	                            // ==============================================================================
	                            // Segment [9]
	                            // ==============================================================================
	                            #tempCalAcc[9] := #tempJerk[9 - 1] * #tempX[9 - 1] + #tempCalAcc[9 - 1];
	                            #tempCalVel[9] := #tempJerk[9 - 1] * #tempX[9 - 1] * #tempX[9 - 1] / 2.0 + #tempCalAcc[9 - 1] * #tempX[9 - 1] + #tempCalVel[9 - 1];
	                            #tempCalPos[9] := #tempJerk[9 - 1] * #tempX[9 - 1] * #tempX[9 - 1] * #tempX[9 - 1] / 6.0 + #tempCalAcc[9 - 1] * #tempX[9 - 1] * #tempX[9 - 1] / 2.0 + #tempCalVel[9 - 1] * #tempX[9 - 1] + #tempCalPos[9 - 1];
	                            IF ABS_LREAL(#tempCalVel[9]) < 0.000000001 THEN
	                                #tempCalVel[9] := 0.0;
	                            END_IF;
	                            IF ABS_LREAL(#tempCalPos[9]) < 0.000000001 THEN
	                                #tempCalPos[9] := 0.0;
	                            END_IF;
	                            #tempA3[9] := #tempJerk[9] / 6.0;
	                            #tempA2[9] := #tempCalAcc[9] / 2.0;
	                            #tempA1[9] := #tempCalVel[9];
	                            #tempA0[9] := #tempCalPos[9];
	                            #tempCam^.Segment[9].a0 := #tempA0[9];
	                            #tempCam^.Segment[9].a1 := #tempA1[9];
	                            #tempCam^.Segment[9].a2 := #tempA2[9];
	                            #tempCam^.Segment[9].a3 := #tempA3[9];
	                            #tempCam^.Segment[9].a4 := 0.0;
	                            #tempCam^.Segment[9].a5 := 0.0;
	                            #tempCam^.Segment[9].a6 := 0.0;
	                            #tempCam^.Segment[9].xmax := #tempCam^.Segment[9 - 1].xmax + #tempX[9];
	                            #tempCam^.Segment[9].xmin := #tempCam^.Segment[9 - 1].xmax;
	                            #tempCam^.Segment[9].sineAmplitude := 0.0;
	                            #tempCam^.Segment[9].sinePeriod := 0.0;
	                            #tempCam^.Segment[9].sinePhase := 0.0;
	                            IF #tempX[9] = 0.0 THEN
	                                #tempCam^.ValidSegment[9] := FALSE;
	                            ELSE
	                                #tempCam^.ValidSegment[9] := TRUE;
	                            END_IF;

	                            // ==============================================================================
	                            // Segment [10]
	                            // ==============================================================================
	                            #tempCalAcc[10] := #tempJerk[10 - 1] * #tempX[10 - 1] + #tempCalAcc[10 - 1];
	                            #tempCalVel[10] := #tempJerk[10 - 1] * #tempX[10 - 1] * #tempX[10 - 1] / 2.0 + #tempCalAcc[10 - 1] * #tempX[10 - 1] + #tempCalVel[10 - 1];
	                            #tempCalPos[10] := #tempJerk[10 - 1] * #tempX[10 - 1] * #tempX[10 - 1] * #tempX[10 - 1] / 6.0 + #tempCalAcc[10 - 1] * #tempX[10 - 1] * #tempX[10 - 1] / 2.0 + #tempCalVel[10 - 1] * #tempX[10 - 1] + #tempCalPos[10 - 1];
	                            IF ABS_LREAL(#tempCalVel[10]) < 0.000000001 THEN
	                                #tempCalVel[10] := 0.0;
	                            END_IF;
	                            IF ABS_LREAL(#tempCalPos[10]) < 0.000000001 THEN
	                                #tempCalPos[10] := 0.0;
	                            END_IF;
	                            #tempA3[10] := #tempJerk[10] / 6.0;
	                            #tempA2[10] := #tempCalAcc[10] / 2.0;
	                            #tempA1[10] := #tempCalVel[10];
	                            #tempA0[10] := #tempCalPos[10];
	                            #tempCam^.Segment[10].a0 := #tempA0[10];
	                            #tempCam^.Segment[10].a1 := #tempA1[10];
	                            #tempCam^.Segment[10].a2 := #tempA2[10];
	                            #tempCam^.Segment[10].a3 := #tempA3[10];
	                            #tempCam^.Segment[10].a4 := 0.0;
	                            #tempCam^.Segment[10].a5 := 0.0;
	                            #tempCam^.Segment[10].a6 := 0.0;
	                            #tempCam^.Segment[10].xmax := #tempCam^.Segment[10 - 1].xmax + #tempX[10];
	                            #tempCam^.Segment[10].xmin := #tempCam^.Segment[10 - 1].xmax;
	                            #tempCam^.Segment[10].sineAmplitude := 0.0;
	                            #tempCam^.Segment[10].sinePeriod := 0.0;
	                            #tempCam^.Segment[10].sinePhase := 0.0;
	                            IF #tempX[10] = 0.0 THEN
	                                #tempCam^.ValidSegment[10] := FALSE;
	                            ELSE
	                                #tempCam^.ValidSegment[10] := TRUE;
	                            END_IF;

	                            // ==============================================================================
	                            // Segment [11]
	                            // ==============================================================================
	                            #tempCalAcc[11] := #tempJerk[11 - 1] * #tempX[11 - 1] + #tempCalAcc[11 - 1];
	                            #tempCalVel[11] := #tempJerk[11 - 1] * #tempX[11 - 1] * #tempX[11 - 1] / 2.0 + #tempCalAcc[11 - 1] * #tempX[11 - 1] + #tempCalVel[11 - 1];
	                            #tempCalPos[11] := #tempJerk[11 - 1] * #tempX[11 - 1] * #tempX[11 - 1] * #tempX[11 - 1] / 6.0 + #tempCalAcc[11 - 1] * #tempX[11 - 1] * #tempX[11 - 1] / 2.0 + #tempCalVel[11 - 1] * #tempX[11 - 1] + #tempCalPos[11 - 1];
	                            IF ABS_LREAL(#tempCalVel[11]) < 0.000000001 THEN
	                                #tempCalVel[11] := 0.0;
	                            END_IF;
	                            IF ABS_LREAL(#tempCalPos[11]) < 0.000000001 THEN
	                                #tempCalPos[11] := 0.0;
	                            END_IF;
	                            #tempA3[11] := #tempJerk[11] / 6.0;
	                            #tempA2[11] := #tempCalAcc[11] / 2.0;
	                            #tempA1[11] := #tempCalVel[11];
	                            #tempA0[11] := #tempCalPos[11];
	                            #tempCam^.Segment[11].a0 := #tempA0[11];
	                            #tempCam^.Segment[11].a1 := #tempA1[11];
	                            #tempCam^.Segment[11].a2 := #tempA2[11];
	                            #tempCam^.Segment[11].a3 := #tempA3[11];
	                            #tempCam^.Segment[11].a4 := 0.0;
	                            #tempCam^.Segment[11].a5 := 0.0;
	                            #tempCam^.Segment[11].a6 := 0.0;
	                            #tempCam^.Segment[11].xmax := #tempCam^.Segment[11 - 1].xmax + #tempX[11];
	                            #tempCam^.Segment[11].xmin := #tempCam^.Segment[11 - 1].xmax;
	                            #tempCam^.Segment[11].sineAmplitude := 0.0;
	                            #tempCam^.Segment[11].sinePeriod := 0.0;
	                            #tempCam^.Segment[11].sinePhase := 0.0;
	                            IF #tempX[11] = 0.0 THEN
	                                #tempCam^.ValidSegment[11] := FALSE;
	                            ELSE
	                                #tempCam^.ValidSegment[11] := TRUE;
	                            END_IF;

	                            // ==============================================================================
	                            // Segment [12]
	                            // ==============================================================================
	                            #tempCalAcc[12] := #tempJerk[12 - 1] * #tempX[12 - 1] + #tempCalAcc[12 - 1];
	                            #tempCalVel[12] := #tempJerk[12 - 1] * #tempX[12 - 1] * #tempX[12 - 1] / 2.0 + #tempCalAcc[12 - 1] * #tempX[12 - 1] + #tempCalVel[12 - 1];
	                            #tempCalPos[12] := #tempJerk[12 - 1] * #tempX[12 - 1] * #tempX[12 - 1] * #tempX[12 - 1] / 6.0 + #tempCalAcc[12 - 1] * #tempX[12 - 1] * #tempX[12 - 1] / 2.0 + #tempCalVel[12 - 1] * #tempX[12 - 1] + #tempCalPos[12 - 1];
	                            IF ABS_LREAL(#tempCalVel[12]) < 0.000000001 THEN
	                                #tempCalVel[12] := 0.0;
	                            END_IF;
	                            IF ABS_LREAL(#tempCalPos[12]) < 0.000000001 THEN
	                                #tempCalPos[12] := 0.0;
	                            END_IF;
	                            #tempA3[12] := #tempJerk[12] / 6.0;
	                            #tempA2[12] := #tempCalAcc[12] / 2.0;
	                            #tempA1[12] := #tempCalVel[12];
	                            #tempA0[12] := #tempCalPos[12];
	                            #tempCam^.Segment[12].a0 := #tempA0[12];
	                            #tempCam^.Segment[12].a1 := #tempA1[12];
	                            #tempCam^.Segment[12].a2 := #tempA2[12];
	                            #tempCam^.Segment[12].a3 := #tempA3[12];
	                            #tempCam^.Segment[12].a4 := 0.0;
	                            #tempCam^.Segment[12].a5 := 0.0;
	                            #tempCam^.Segment[12].a6 := 0.0;
	                            #tempCam^.Segment[12].xmax := #tempCam^.Segment[12 - 1].xmax + #tempX[12];
	                            #tempCam^.Segment[12].xmin := #tempCam^.Segment[12 - 1].xmax;
	                            #tempCam^.Segment[12].sineAmplitude := 0.0;
	                            #tempCam^.Segment[12].sinePeriod := 0.0;
	                            #tempCam^.Segment[12].sinePhase := 0.0;
	                            IF #tempX[12] = 0.0 THEN
	                                #tempCam^.ValidSegment[12] := FALSE;
	                            ELSE
	                                #tempCam^.ValidSegment[12] := TRUE;
	                            END_IF;

	                            // ==============================================================================
	                            // Segment [13]
	                            // ==============================================================================
	                            #tempCalAcc[13] := #tempJerk[13 - 1] * #tempX[13 - 1] + #tempCalAcc[13 - 1];
	                            #tempCalVel[13] := #tempJerk[13 - 1] * #tempX[13 - 1] * #tempX[13 - 1] / 2.0 + #tempCalAcc[13 - 1] * #tempX[13 - 1] + #tempCalVel[13 - 1];
	                            #tempCalPos[13] := #tempJerk[13 - 1] * #tempX[13 - 1] * #tempX[13 - 1] * #tempX[13 - 1] / 6.0 + #tempCalAcc[13 - 1] * #tempX[13 - 1] * #tempX[13 - 1] / 2.0 + #tempCalVel[13 - 1] * #tempX[13 - 1] + #tempCalPos[13 - 1];
	                            IF ABS_LREAL(#tempCalVel[13]) < 0.000000001 THEN
	                                #tempCalVel[13] := 0.0;
	                            END_IF;
	                            IF ABS_LREAL(#tempCalPos[13]) < 0.000000001 THEN
	                                #tempCalPos[13] := 0.0;
	                            END_IF;
	                            #tempA3[13] := #tempJerk[13] / 6.0;
	                            #tempA2[13] := #tempCalAcc[13] / 2.0;
	                            #tempA1[13] := #tempCalVel[13];
	                            #tempA0[13] := #tempCalPos[13];
	                            #tempCam^.Segment[13].a0 := #tempA0[13];
	                            #tempCam^.Segment[13].a1 := #tempA1[13];
	                            #tempCam^.Segment[13].a2 := #tempA2[13];
	                            #tempCam^.Segment[13].a3 := #tempA3[13];
	                            #tempCam^.Segment[13].a4 := 0.0;
	                            #tempCam^.Segment[13].a5 := 0.0;
	                            #tempCam^.Segment[13].a6 := 0.0;
	                            #tempCam^.Segment[13].xmax := #tempCam^.Segment[13 - 1].xmax + #tempX[13];
	                            #tempCam^.Segment[13].xmin := #tempCam^.Segment[13 - 1].xmax;
	                            #tempCam^.Segment[13].sineAmplitude := 0.0;
	                            #tempCam^.Segment[13].sinePeriod := 0.0;
	                            #tempCam^.Segment[13].sinePhase := 0.0;
	                            IF #tempX[13] = 0.0 THEN
	                                #tempCam^.ValidSegment[13] := FALSE;
	                            ELSE
	                                #tempCam^.ValidSegment[13] := TRUE;
	                            END_IF;

	                            // ==============================================================================
	                            // Segment [14]
	                            // ==============================================================================
	                            #tempCalAcc[14] := #tempJerk[14 - 1] * #tempX[14 - 1] + #tempCalAcc[14 - 1];
	                            #tempCalVel[14] := #tempJerk[14 - 1] * #tempX[14 - 1] * #tempX[14 - 1] / 2.0 + #tempCalAcc[14 - 1] * #tempX[14 - 1] + #tempCalVel[14 - 1];
	                            #tempCalPos[14] := #tempJerk[14 - 1] * #tempX[14 - 1] * #tempX[14 - 1] * #tempX[14 - 1] / 6.0 + #tempCalAcc[14 - 1] * #tempX[14 - 1] * #tempX[14 - 1] / 2.0 + #tempCalVel[14 - 1] * #tempX[14 - 1] + #tempCalPos[14 - 1];
	                            IF ABS_LREAL(#tempCalVel[14]) < 0.000000001 THEN
	                                #tempCalVel[14] := 0.0;
	                            END_IF;
	                            IF ABS_LREAL(#tempCalPos[14]) < 0.000000001 THEN
	                                #tempCalPos[14] := 0.0;
	                            END_IF;
	                            #tempA3[14] := #tempJerk[14] / 6.0;
	                            #tempA2[14] := #tempCalAcc[14] / 2.0;
	                            #tempA1[14] := #tempCalVel[14];
	                            #tempA0[14] := #tempCalPos[14];
	                            #tempCam^.Segment[14].a0 := #tempA0[14];
	                            #tempCam^.Segment[14].a1 := #tempA1[14];
	                            #tempCam^.Segment[14].a2 := #tempA2[14];
	                            #tempCam^.Segment[14].a3 := #tempA3[14];
	                            #tempCam^.Segment[14].a4 := 0.0;
	                            #tempCam^.Segment[14].a5 := 0.0;
	                            #tempCam^.Segment[14].a6 := 0.0;
	                            #tempCam^.Segment[14].xmax := #tempCam^.Segment[14 - 1].xmax + #tempX[14];
	                            #tempCam^.Segment[14].xmin := #tempCam^.Segment[14 - 1].xmax;
	                            #tempCam^.Segment[14].sineAmplitude := 0.0;
	                            #tempCam^.Segment[14].sinePeriod := 0.0;
	                            #tempCam^.Segment[14].sinePhase := 0.0;
	                            IF #tempX[14] = 0.0 THEN
	                                #tempCam^.ValidSegment[14] := FALSE;
	                            ELSE
	                                #tempCam^.ValidSegment[14] := TRUE;
	                            END_IF;

	                            // ==============================================================================
	                            // Segment [15]
	                            // ==============================================================================
	                            #tempCalAcc[15] := #tempJerk[15 - 1] * #tempX[15 - 1] + #tempCalAcc[15 - 1];
	                            #tempCalVel[15] := #tempJerk[15 - 1] * #tempX[15 - 1] * #tempX[15 - 1] / 2.0 + #tempCalAcc[15 - 1] * #tempX[15 - 1] + #tempCalVel[15 - 1];
	                            #tempCalPos[15] := #tempJerk[15 - 1] * #tempX[15 - 1] * #tempX[15 - 1] * #tempX[15 - 1] / 6.0 + #tempCalAcc[15 - 1] * #tempX[15 - 1] * #tempX[15 - 1] / 2.0 + #tempCalVel[15 - 1] * #tempX[15 - 1] + #tempCalPos[15 - 1];
	                            IF ABS_LREAL(#tempCalVel[15]) < 0.000000001 THEN
	                                #tempCalVel[15] := 0.0;
	                            END_IF;
	                            IF ABS_LREAL(#tempCalPos[15]) < 0.000000001 THEN
	                                #tempCalPos[15] := 0.0;
	                            END_IF;
	                            #tempA3[15] := #tempJerk[15] / 6.0;
	                            #tempA2[15] := #tempCalAcc[15] / 2.0;
	                            #tempA1[15] := #tempCalVel[15];
	                            #tempA0[15] := #tempCalPos[15];
	                            #tempCam^.Segment[15].a0 := #tempA0[15];
	                            #tempCam^.Segment[15].a1 := #tempA1[15];
	                            #tempCam^.Segment[15].a2 := #tempA2[15];
	                            #tempCam^.Segment[15].a3 := #tempA3[15];
	                            #tempCam^.Segment[15].a4 := 0.0;
	                            #tempCam^.Segment[15].a5 := 0.0;
	                            #tempCam^.Segment[15].a6 := 0.0;
	                            #tempCam^.Segment[15].xmax := #tempCam^.Segment[15 - 1].xmax + #tempX[15];
	                            #tempCam^.Segment[15].xmin := #tempCam^.Segment[15 - 1].xmax;
	                            #tempCam^.Segment[15].sineAmplitude := 0.0;
	                            #tempCam^.Segment[15].sinePeriod := 0.0;
	                            #tempCam^.Segment[15].sinePhase := 0.0;
	                            IF #tempX[15] = 0.0 THEN
	                                #tempCam^.ValidSegment[15] := FALSE;
	                            ELSE
	                                #tempCam^.ValidSegment[15] := TRUE;
	                            END_IF;

	                            // ==============================================================================
	                            // Segment [16]
	                            // ==============================================================================
	                            #tempCalAcc[16] := #tempJerk[16 - 1] * #tempX[16 - 1] + #tempCalAcc[16 - 1];
	                            #tempCalVel[16] := #tempJerk[16 - 1] * #tempX[16 - 1] * #tempX[16 - 1] / 2.0 + #tempCalAcc[16 - 1] * #tempX[16 - 1] + #tempCalVel[16 - 1];
	                            #tempCalPos[16] := #tempJerk[16 - 1] * #tempX[16 - 1] * #tempX[16 - 1] * #tempX[16 - 1] / 6.0 + #tempCalAcc[16 - 1] * #tempX[16 - 1] * #tempX[16 - 1] / 2.0 + #tempCalVel[16 - 1] * #tempX[16 - 1] + #tempCalPos[16 - 1];
	                            IF ABS_LREAL(#tempCalVel[16]) < 0.000000001 THEN
	                                #tempCalVel[16] := 0.0;
	                            END_IF;
	                            IF ABS_LREAL(#tempCalPos[16]) < 0.000000001 THEN
	                                #tempCalPos[16] := 0.0;
	                            END_IF;
	                            #tempA3[16] := #tempJerk[16] / 6.0;
	                            #tempA2[16] := #tempCalAcc[16] / 2.0;
	                            #tempA1[16] := #tempCalVel[16];
	                            #tempA0[16] := #tempCalPos[16];
	                            #tempCam^.Segment[16].a0 := #tempA0[16];
	                            #tempCam^.Segment[16].a1 := #tempA1[16];
	                            #tempCam^.Segment[16].a2 := #tempA2[16];
	                            #tempCam^.Segment[16].a3 := #tempA3[16];
	                            #tempCam^.Segment[16].a4 := 0.0;
	                            #tempCam^.Segment[16].a5 := 0.0;
	                            #tempCam^.Segment[16].a6 := 0.0;
	                            #tempCam^.Segment[16].xmax := #tempCam^.Segment[16 - 1].xmax + #tempX[16];
	                            #tempCam^.Segment[16].xmin := #tempCam^.Segment[16 - 1].xmax;
	                            #tempCam^.Segment[16].sineAmplitude := 0.0;
	                            #tempCam^.Segment[16].sinePeriod := 0.0;
	                            #tempCam^.Segment[16].sinePhase := 0.0;
	                            IF #tempX[16] = 0.0 THEN
	                                #tempCam^.ValidSegment[16] := FALSE;
	                            ELSE
	                                #tempCam^.ValidSegment[16] := TRUE;
	                            END_IF;
	                        END_REGION
	                    END_REGION

	                END_IF;
	                #statEndTime := TIME_TCK();
	                #statTimeTable[#CC_CALCULATE] := #statEndTime - #statStartTime;
	                #statStartTime := TIME_TCK();
	                #statCalculateCamState := #CC_INTERPOLATE;
	            END_REGION

	        #CC_INTERPOLATE:
	            REGION INTERPOLATE
	                IF #instMCInterpolateCam.Done
	                THEN
	                    #statEndTime := TIME_TCK();
	                    #statTimeTable[#CC_INTERPOLATE] := #statEndTime - #statStartTime;
	                    #statStartTime := TIME_TCK();
	                    #statCalculateCamState := #CC_DONE;
	                END_IF;
	            END_REGION

	        #CC_DONE:
	            REGION DONE
	                ;
	            END_REGION

	        #CC_ERROR:
	            REGION ERROR
	                ;
	            END_REGION
	    END_CASE;
	END_REGION

	REGION Instance
	    #instMCInterpolateCam(Cam := #tempCam^,
	                          Execute := #statCalculateCamState = #CC_INTERPOLATE);
	    #instMCCopyCamData(Cam := #tempCam^,
	                       Execute := #statCalculateCamState = #CC_INITIALIZE1 OR #statCalculateCamState = #CC_INITIALIZE3,
	                       Mode := 0,
	                       StartPointCam := 1,
	                       StartSegmentCam := 1,
	                       StartPointArray := 1,
	                       StartSegmentArray := 1,
	                       ArrayOfPoints := #EmptyPoint,
	                       ArrayOfSegments := #EmptySegment);
	END_REGION

	REGION Outputs
	    #busy := #statCalculateCamState = #CC_INITIALIZE1
	    OR #statCalculateCamState = #CC_INITIALIZE2
	    OR #statCalculateCamState = #CC_INITIALIZE3
	    OR #statCalculateCamState = #CC_CALCULATE
	    OR #statCalculateCamState = #CC_INTERPOLATE;
	    #error := #statCalculateCamState = #CC_ERROR;
	    #done := #statCalculateCamState = #CC_DONE;
	END_REGION
END_FUNCTION_BLOCK

